Staubli VAL3: stop.pgx

program stop()
begin
  popUpMsg("Pending movement commands have been canceled")
  resetMotion()
end
